Omron Sysmac Studio project stopwatch (Sysmac Studio 1.60.0.64010, StandardProject)

# Controller cpu: NX1P2-1040DT1 version 1.64
Task PrimaryTask (priority 4, period or condition 2000): Program0

TYPE My_sw : STRUCT
    hours : INT;
    min : INT;
    sec : INT;
    start_stop : BOOL;
    reset : BOOL;
END_STRUCT END_TYPE

VAR_GLOBAL
    Stopwatch_tag : My_sw;
    one_sec : BOOL;
END_VAR

PROGRAM Program0
VAR
    r_trigg : R_TRIG;
    r_trigg1 : R_TRIG;
END_VAR
VAR_EXTERNAL
    one_sec : BOOL;
    Stopwatch_tag : My_sw;
END_VAR
VAR
    _p1 : BOOL;
    _p2 : BOOL;
    _p3 : BOOL;
END_VAR

(* Section stopwatch: ladder, written here as Structured Text *)

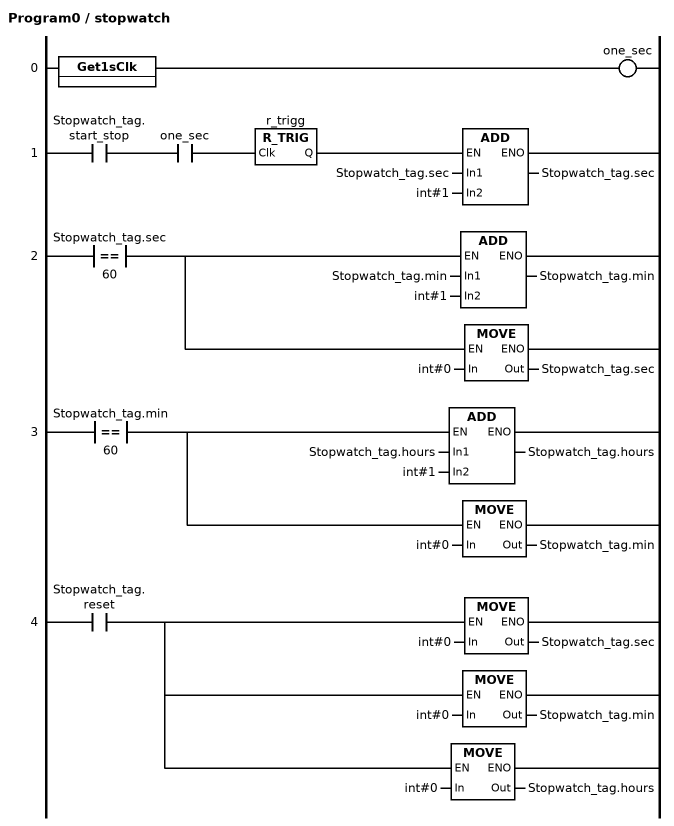
(* Rung 0 *)
one_sec := Get1sClk();
(* Rung 1 *)
r_trigg(Clk := Stopwatch_tag.start_stop AND one_sec);
IF r_trigg.Q THEN Stopwatch_tag.sec := Stopwatch_tag.sec + int#1; END_IF;
(* Rung 2 *)
_p1 := Stopwatch_tag.sec = 60;
IF _p1 THEN
    Stopwatch_tag.min := Stopwatch_tag.min + int#1;
    Stopwatch_tag.sec := int#0;
END_IF;
(* Rung 3 *)
_p2 := Stopwatch_tag.min = 60;
IF _p2 THEN
    Stopwatch_tag.hours := Stopwatch_tag.hours + int#1;
    Stopwatch_tag.min := int#0;
END_IF;
(* Rung 4 *)
_p3 := Stopwatch_tag.reset;
IF _p3 THEN
    Stopwatch_tag.sec := int#0;
    Stopwatch_tag.min := int#0;
    Stopwatch_tag.hours := int#0;
END_IF;
END_PROGRAM

# Device HMI_NA5_0 (NA): not converted